# EPICS autosave request: pmac/pmacCsController_settings.req
$(PMAC):CS$(CS):CsMoveTime
